FUNCTION_BLOCK "EM_TransferDischarge"
{ S7_Optimized_Access := 'TRUE' }


BEGIN

END_FUNCTION_BLOCK
